FUNCTION fc_Year_Of_Date : INT
VAR_INPUT
		IDATE : DATE;
END_VAR
VAR
END_VAR

fc_Year_Of_Date := DWORD_TO_INT((DATE_TO_DWORD(idate) + 43200) / 31557600 + 1970);

END_FUNCTION

(* stored: Version 1.1.0.1, ProductVersion 3.1.4024.11
   POU fc_Year_Of_Date: Id {e6ce8169-2218-4c59-b394-d4f682f27f31}, SpecialFunc None *)
